(* PLC project prj, KAIST_DSLAB noNameNow 1, author bwkim *)
(* stored: creationDateTime 2015-7-21T04:57:22, modificationDateTime 2015-7-21T04:57:22 *)

PROGRAM program4____sub1
  VAR
    MF_PTRIP_TON : null;
  END_VAR
  VAR
    MF_TRIP_TON : null;
  END_VAR
  VAR_IN_OUT
    TRIP : BOOL := FALSE;
  END_VAR
  VAR_IN_OUT
    PTRIP_LOGIC : BOOL := FALSE;
  END_VAR
  VAR_IN_OUT
    TRIP_LOGIC : BOOL := FALSE;
  END_VAR
  VAR_IN_OUT
    PTRIP : BOOL := FALSE;
  END_VAR
  VAR  (* added by the conversion: wires and edge detectors of the diagram *)
    _SEL_REAL70_OUT : ANY;
    _SEL_REAL53_OUT : ANY;
    _SEL_REAL54_OUT : ANY;
    _SEL_REAL71_OUT : ANY;
    _SEL_BOOL83_OUT : BOOL;
    _SEL_REAL39_OUT : ANY;
    _SEL_BOOL89_OUT : BOOL;
    _SEL_REAL90_OUT : ANY;
    _AND2_BOOL64_OUT : BOOL;
    _SEL_REAL97_OUT : ANY;
    _SEL_REAL98_OUT : ANY;
    _AND2_BOOL66_OUT : ANY;
  END_VAR

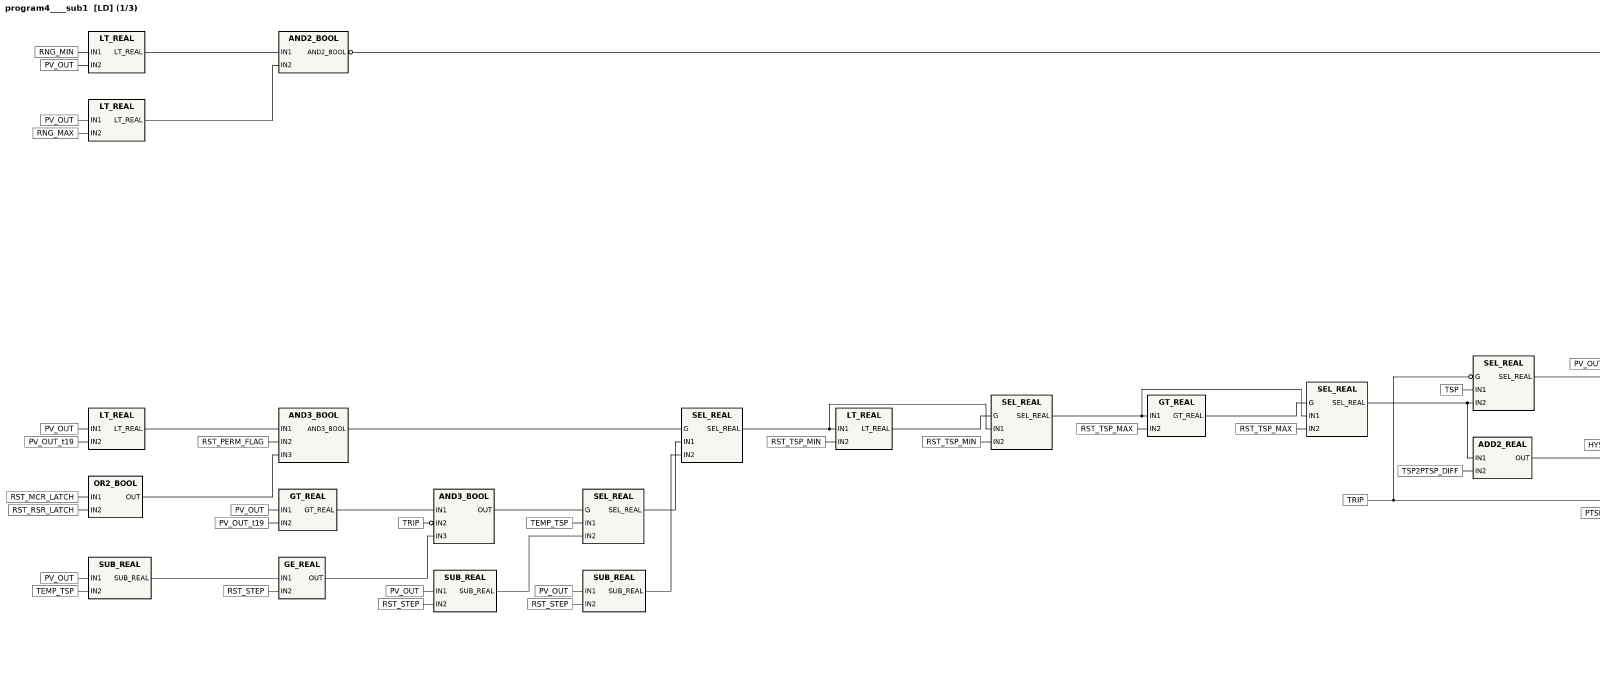
(* LD diagram, written out as Structured Text *)
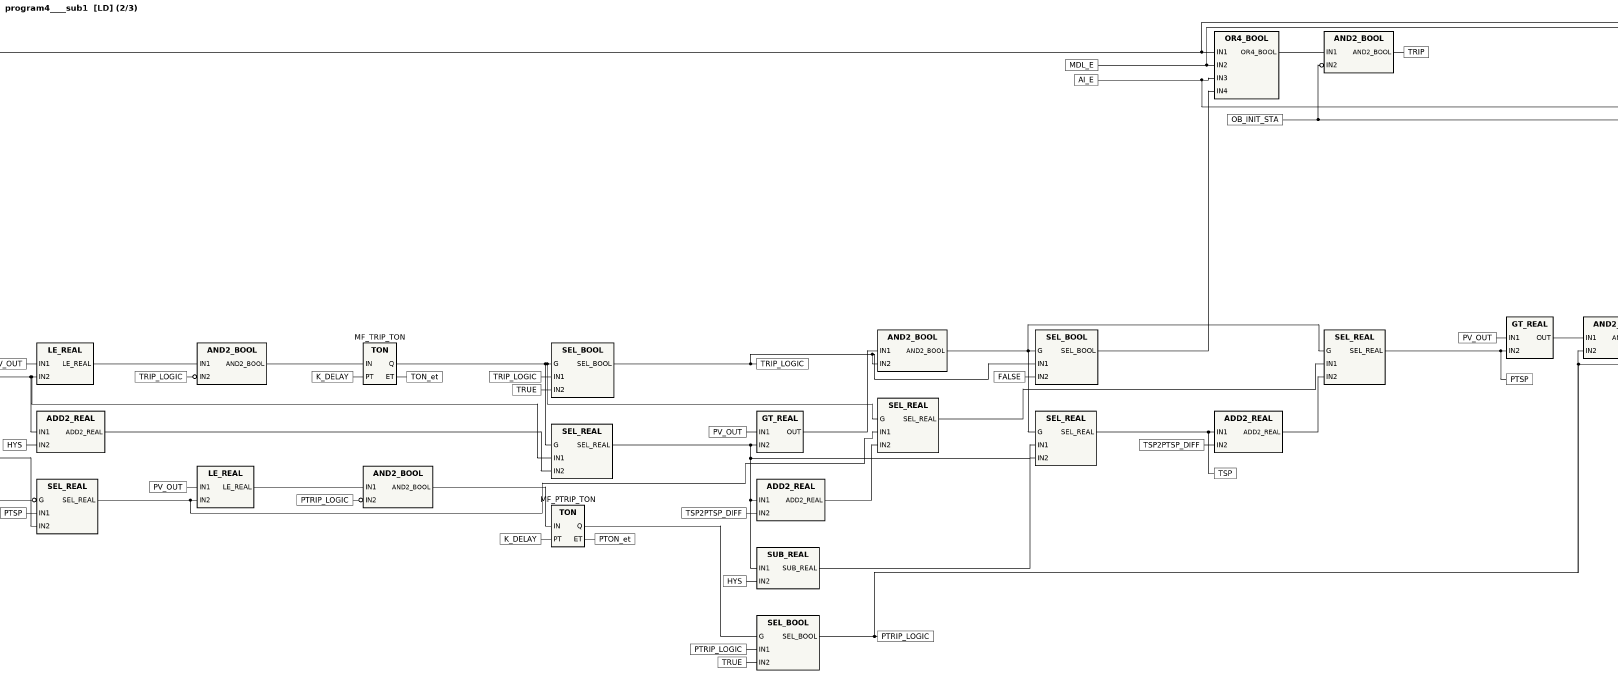
_SEL_REAL70_OUT := SEL_REAL(AND3_BOOL(LT_REAL(PV_OUT, PV_OUT_t19), RST_PERM_FLAG, OR2_BOOL(RST_MCR_LATCH, RST_RSR_LATCH)), SEL_REAL(AND3_BOOL(GT_REAL(PV_OUT, PV_OUT_t19), NOT TRIP, GE_REAL(SUB_REAL(PV_OUT, TEMP_TSP), RST_STEP)), TEMP_TSP, SUB_REAL(PV_OUT, RST_STEP)), SUB_REAL(PV_OUT, RST_STEP));
_SEL_REAL53_OUT := SEL_REAL(LT_REAL(_SEL_REAL70_OUT, RST_TSP_MIN), _SEL_REAL70_OUT, RST_TSP_MIN);
_SEL_REAL54_OUT := SEL_REAL(GT_REAL(_SEL_REAL53_OUT, RST_TSP_MAX), _SEL_REAL53_OUT, RST_TSP_MAX);
_SEL_REAL71_OUT := SEL_REAL(NOT TRIP, PTSP, ADD2_REAL(_SEL_REAL54_OUT, TSP2PTSP_DIFF));
MF_PTRIP_TON(IN := AND2_BOOL(LE_REAL(PV_OUT, _SEL_REAL71_OUT), NOT PTRIP_LOGIC), PT := K_DELAY);
_SEL_BOOL83_OUT := SEL_BOOL(MF_PTRIP_TON.Q, PTRIP_LOGIC, TRUE);
PTRIP_LOGIC := _SEL_BOOL83_OUT;
PTON_et := MF_PTRIP_TON.ET;
_SEL_REAL39_OUT := SEL_REAL(NOT TRIP, TSP, _SEL_REAL54_OUT);
MF_TRIP_TON(IN := AND2_BOOL(LE_REAL(PV_OUT, _SEL_REAL39_OUT), NOT TRIP_LOGIC), PT := K_DELAY);
_SEL_BOOL89_OUT := SEL_BOOL(MF_TRIP_TON.Q, TRIP_LOGIC, TRUE);
TRIP_LOGIC := _SEL_BOOL89_OUT;
TON_et := MF_TRIP_TON.ET;
_SEL_REAL90_OUT := SEL_REAL(MF_TRIP_TON.Q, _SEL_REAL39_OUT, ADD2_REAL(_SEL_REAL39_OUT, HYS));
_AND2_BOOL64_OUT := AND2_BOOL(GT_REAL(PV_OUT, _SEL_REAL90_OUT), _SEL_BOOL89_OUT);
_SEL_REAL97_OUT := SEL_REAL(_AND2_BOOL64_OUT, _SEL_REAL90_OUT, SUB_REAL(_SEL_REAL90_OUT, HYS));
TSP := _SEL_REAL97_OUT;
_SEL_REAL98_OUT := SEL_REAL(_AND2_BOOL64_OUT, SEL_REAL(MF_TRIP_TON.Q, _SEL_REAL71_OUT, ADD2_REAL(_SEL_REAL90_OUT, TSP2PTSP_DIFF)), ADD2_REAL(_SEL_REAL97_OUT, TSP2PTSP_DIFF));
PTSP := _SEL_REAL98_OUT;
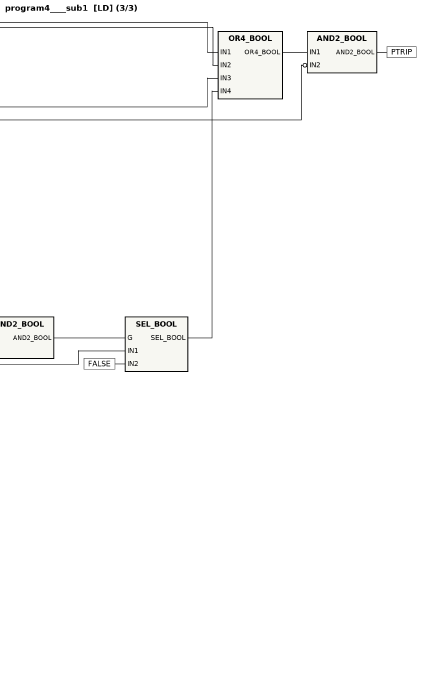
_AND2_BOOL66_OUT := AND2_BOOL(LT_REAL(RNG_MIN, PV_OUT), LT_REAL(PV_OUT, RNG_MAX));
PTRIP := AND2_BOOL(OR4_BOOL(_AND2_BOOL66_OUT, MDL_E, AI_E, SEL_BOOL(AND2_BOOL(GT_REAL(PV_OUT, _SEL_REAL98_OUT), _SEL_BOOL83_OUT), _SEL_BOOL83_OUT, FALSE)), NOT OB_INIT_STA);
TRIP := AND2_BOOL(OR4_BOOL(_AND2_BOOL66_OUT, MDL_E, AI_E, SEL_BOOL(_AND2_BOOL64_OUT, _SEL_BOOL89_OUT, FALSE)), NOT OB_INIT_STA);
END_PROGRAM
